INTERFACE Name

{attribute 'monitoring' := 'call'}
PROPERTY Name : T_MaxString
GET
END_GET
SET
END_SET
END_PROPERTY

END_INTERFACE

(* stored: Version 1.1.0.1
   Itf Name: Id {fc4be3a0-9295-0d76-0cd4-c8f5c6544e2f}
   Property Name: Id {4aed2bca-5d35-04a5-10f7-74ad509dbcf2}
   Get Get: Id {92af3c9b-98b2-0cf2-3701-7d1dda325c3a}
   Set Set: Id {b5ca13f9-2b56-0775-0301-98fbfef773c5} *)
